Yaskawa INFORM job: OK_R2_O50&56(110_90,0)AWOK.JBI

/JOB
//NAME OK_R2_O50&56(110_90,0)AWOK
///FOLDERNAME X4
//POS
///NPOS 267,267,267,15,0,0
///TOOL 0
///POSTYPE PULSE
///PULSE
C00000=174960,-106597,-120103,3797,95090,-7084
C00001=145956,12891,-49012,9197,114627,-15113
C00002=146175,14682,13914,33266,91894,-54167
C00003=181880,-35169,-29211,31591,75181,-62241
C00004=185949,-21647,605,33162,63920,-63937
C00005=185949,-19989,4400,33558,62671,-64348
C00006=185949,-21647,605,33162,63920,-63937
C00007=186497,-22505,-4,33104,63655,-63786
C00008=185949,-21647,605,33162,63920,-63937
C00009=186993,-19461,2175,32975,63654,-63571
C00010=187282,-18335,3806,33046,63184,-63596
C00011=186993,-19461,2175,32975,63654,-63571
C00012=174899,-22090,-15041,32767,76141,-64809
C00013=150915,-27906,-19346,34122,85374,-71784
C00014=124603,-47737,-34158,-19131,104982,62056
C00015=121442,-51513,-32422,-19687,101389,61480
C00016=118855,-51471,-32397,-20347,100766,60636
C00017=118855,-50574,-30118,-20274,99880,60787
C00018=118855,-51471,-32397,-20347,100766,60636
C00019=121442,-51513,-32422,-19687,101389,61480
C00020=121797,-50324,-29168,-19487,100158,61813
C00021=120620,-50331,-29171,-19792,99877,61431
C00022=121797,-50324,-29168,-19487,100158,61813
C00023=121442,-51513,-32422,-19687,101389,61480
C00024=121603,-51176,-29855,-19536,100099,61752
C00025=121615,-53238,-31000,-19508,99766,61811
C00026=121603,-51176,-29855,-19536,100099,61752
C00027=122128,-47866,-34232,-19785,104374,61232
C00028=84141,-29178,-36607,-14646,114104,67707
C00029=82791,-33286,-36430,-14724,111710,67503
C00030=82229,-34853,-36282,-14765,110740,67415
C00031=82178,-34515,-34630,-14688,109914,67503
C00032=82229,-34853,-36282,-14765,110740,67415
C00033=79147,-30434,-31070,-15425,109262,66446
C00034=78452,-32631,-32544,-15567,108914,66232
C00035=79147,-30434,-31070,-15425,109262,66446
C00036=79730,-28966,-31252,-15378,110209,66539
C00037=81132,-25108,-31519,-15285,112547,66756
C00038=130185,-45166,-65053,-10858,92991,77597
C00039=107206,26705,4589,-9987,92468,27814
C00040=98659,45218,28508,-8039,93095,24888
C00041=98424,43781,30134,-8022,91351,24920
C00042=98486,43736,30153,-8021,91323,24943
C00043=98486,44012,31621,-8015,90571,24990
C00044=98486,43353,27835,-8034,92544,24864
C00045=106492,38043,26451,-21991,88874,27615
C00046=105786,38474,26895,-21964,88638,27404
C00047=106495,38155,26700,-21991,88785,27632
C00048=106495,37420,22299,-22016,90954,27236
C00049=111541,35328,25383,-22123,89542,29330
C00050=102045,-19807,-16561,-21845,84655,26763
C00051=74840,-13391,-38223,-2617,97503,17820
C00052=66507,5010,-12577,6934,97902,16018
C00053=66741,4651,-9261,6890,95673,15973
C00054=66101,6043,-7102,6886,95120,15724
C00055=66101,6129,-6115,6879,94563,15693
C00056=66101,5877,-9999,6916,96808,15817
C00057=80836,-17286,-23478,-14204,80508,20001
C00058=80064,-16344,-22775,-14064,80424,19740
C00059=80850,-17465,-25526,-14169,81645,19874
C00060=68799,5840,-15749,112,106098,15895
C00061=55050,-26211,-40797,-896,104976,11120
C00062=53240,-26394,-33808,-1003,100562,10527
C00063=53174,-26119,-32540,-1008,99922,10509
C00064=53174,-26003,-31510,-1007,99347,10512
C00065=53450,-26813,-34326,-989,100667,10598
C00066=66076,-50527,-45741,-15470,82986,15464
C00067=65365,-49438,-45112,-15396,83017,15209
C00068=66444,-51488,-48366,-15481,84138,15447
C00069=76298,-64666,-67677,-16335,90985,18012
C00070=121005,-146046,-93198,-13283,20086,-50099
C00071=121076,-175637,-121627,-12100,22333,-50657
C00072=121076,-175637,-121627,-12100,22333,-50657
C00073=119842,-145846,-119955,19490,98596,44269
C00074=120072,-86643,-91493,20899,110694,78316
C00075=121200,-92303,-90459,20559,107088,78084
C00076=140479,-121048,-96992,20484,87219,81696
C00077=140479,-120457,-95830,20487,86831,81630
C00078=138616,-107413,-91097,21806,95703,82500
C00079=139134,-110877,-92284,21800,94587,82488
C00080=138616,-107413,-91097,21806,95703,82500
C00081=138504,-107678,-93902,21887,97214,82736
C00082=111033,-68243,-79959,15660,119373,68405
C00083=110238,-79863,-86906,15259,112779,67243
C00084=110238,-79955,-85752,15166,112047,67143
C00085=111039,-68171,-79817,15653,119324,68399
C00086=110811,-71611,-81502,15474,118663,68211
C00087=111039,-68171,-79817,15653,119324,68399
C00088=117681,-73428,-89845,994,113898,68956
C00089=117328,-75555,-88746,937,112132,68814
C00090=117314,-76363,-88422,931,111517,68804
C00091=117314,-76477,-87912,929,111141,68802
C00092=117314,-76038,-89659,939,112445,68812
C00093=117225,-80228,-90181,914,110615,68766
C00094=117357,-73687,-89896,955,113798,68838
C00095=117304,-75426,-92745,956,114658,68828
C00096=117163,-75550,-92733,938,114587,68776
C00097=117163,-75975,-91679,932,113721,68770
C00098=117163,-75740,-92281,935,114212,68773
C00099=117065,-80067,-94252,916,113200,68731
C00100=117163,-75740,-92281,935,114212,68773
C00101=126928,-93462,-104099,-21125,97375,56056
C00102=123436,-95743,-101732,-20630,94052,55403
C00103=119720,-93386,-98939,-20195,92672,54328
C00104=119720,-93542,-97538,-20172,91785,54475
C00105=119720,-93459,-98367,-20185,92306,54389
C00106=117930,-93370,-98332,-19971,91899,53827
C00107=119720,-93459,-98367,-20185,92306,54389
C00108=119671,-100746,-101187,-20141,90406,54690
C00109=119720,-93459,-98367,-20185,92306,54389
C00110=121215,-96042,-102269,-20389,93677,54685
C00111=124737,-93931,-104706,-20902,96960,55358
C00112=120615,-97600,-94225,-24394,68229,41312
C00113=121614,-94302,-98325,-24715,72989,35072
C00114=121413,-94319,-98186,-24655,72844,35027
C00115=121413,-94400,-96939,-24754,72105,35186
C00116=121413,-94319,-98186,-24655,72844,35027
C00117=119573,-94306,-98179,-23998,72315,34443
C00118=121413,-94319,-98186,-24655,72844,35027
C00119=131582,-92162,-101045,-27739,78553,37534
C00120=149979,-79190,-101251,-32758,90741,41130
C00121=131734,108486,68329,-27886,77598,37823
C00122=131746,115175,77213,-28093,75801,38268
C00123=128705,103754,56939,-17355,80936,37498
C00124=126391,103513,58781,-16629,79272,36943
C00125=126391,103204,59430,-16657,78740,37018
C00126=126391,103325,59164,-16645,78953,36987
C00127=131461,101888,64135,-32515,75623,37675
C00128=130460,102804,65331,-32242,75027,37451
C00129=132956,104856,68008,-33106,75465,38321
C00130=123747,88520,39161,-14959,81804,36039
C00131=123722,90598,43933,-15013,79993,36251
C00132=123722,90479,44118,-15020,79823,36272
C00133=123708,91557,46446,-15056,78971,36374
C00134=123735,88704,42579,-15029,79860,36272
C00135=122122,90222,44481,-14459,79203,35813
C00136=121873,91643,46282,-14382,78796,35780
C00137=122407,90627,44476,-14554,79458,35880
C00138=127598,110669,63569,-17480,87727,36370
C00139=127458,127775,88290,-17571,81562,37206
C00140=126717,107110,60862,-17217,87970,36047
C00141=121872,67125,15966,-8400,79107,26604
C00142=119947,67807,18007,-7580,78039,26067
C00143=121767,74654,26232,-6383,76292,25284
C00144=123564,69808,18958,-7132,78404,25740
C00145=121169,67878,17908,-8113,78241,26441
C00146=120006,67962,18206,-7608,78000,26088
C00147=117920,61625,14270,-6708,77001,25483
C00148=118781,60315,11658,-7068,77995,25701
C00149=123961,59152,819,-9198,84481,26863
C00150=132618,-110497,-108947,-28734,74981,37704
C00151=124566,-101520,-102656,-26093,73034,35072
C00152=121381,-96484,-98543,-24994,72121,34061
C00153=122368,-97019,-90544,-25347,66960,42290
C00154=120612,-98338,-92224,-24658,66756,41637
C00155=120867,-94519,-89971,-24653,67354,41604
C00156=120867,-94608,-89971,-24661,67311,41612
C00157=126048,-45476,-69322,-31035,100254,58694
C00158=113068,-21387,-59721,-17378,114816,66130
C00159=116612,-26582,-62582,-17226,114626,67431
C00160=116612,-22676,-66743,-18014,118989,66712
C00161=96791,-67830,-88966,-12124,96584,58954
C00162=98008,-71855,-88035,-12234,94161,59592
C00163=126837,-94677,-94277,-15990,96379,69031
C00164=126113,-98665,-96629,-15951,95659,68871
C00165=124903,-86613,-90535,-14366,101584,74527
C00166=124985,-88200,-92279,-14134,101025,73532
C00167=124953,-89747,-92480,-14095,100368,73599
C00168=120613,-99078,-98492,-7508,100072,69302
C00169=121484,-95136,-96163,-7500,100739,69561
C00170=172923,-99546,-90349,-10002,102117,90375
C00171=179538,-101142,-90555,-8602,100288,90316
C00172=174679,-92302,-94882,-9461,106868,88107
C00173=153430,-78772,-107192,1998,100273,82038
C00174=120149,-70168,-111353,20212,74375,72326
C00175=120057,-133921,-120473,34069,36215,62022
C00176=120146,-106815,-117651,27009,46787,66237
C00177=120793,-117832,-87628,5856,54262,-2374
C00178=128370,-47930,-37102,5352,91873,-78331
C00179=120655,-51136,-30966,4745,86952,-81146
C00180=120656,-51126,-30961,4745,86954,-81145
C00181=121240,-72948,-42427,4950,70443,-81585
C00182=120654,-52833,-32998,4744,87329,-81132
C00183=120662,-49043,-29779,4745,87295,-81131
C00184=130317,-72190,-42085,4090,70120,-78412
C00185=120656,-51164,-30982,4745,86947,-81145
C00186=120655,-51174,-30987,4745,86946,-81146
C00187=120663,-45936,-34749,4755,91934,-80956
C00188=120658,-53922,-38518,-13016,106165,78731
C00189=120658,-51068,-30928,-12795,103038,79070
C00190=123140,-68547,-43521,-11941,93024,80951
C00191=120664,-48985,-29748,-12815,103375,79036
C00192=120728,-51718,-32595,-12818,103725,79022
C00193=121911,-67959,-43086,-12159,93263,80503
C00194=120658,-51052,-30919,-12796,103041,79070
C00195=120658,-51066,-30927,-12796,103039,79070
C00196=93952,-51121,-30967,-10241,104523,-67822
C00197=93953,-51118,-30965,-10240,104524,-67822
C00198=95953,-52479,-31764,-9588,104560,-67115
C00199=94418,-49164,-29853,-10109,104897,-67688
C00200=92862,-50813,-31445,-10614,104829,-68238
C00201=95353,-51547,-30566,-9769,104235,-67302
C00202=95660,-51090,-34260,-9806,106744,-67396
C00203=98759,-53921,-36367,-8775,106946,-66293
C00204=98759,-54646,-38349,-8822,107784,-66355
C00205=121493,-81341,-55216,-13751,94719,44592
C00206=118132,-76574,-45148,-14317,90501,43918
C00207=115160,-74416,-40204,-14849,88108,43182
C00208=114252,-83925,-43808,-15028,85362,43206
C00209=116252,-82247,-47187,-14646,88567,43499
C00210=104568,-69110,-41017,-10991,94760,66686
C00211=117881,-67291,-35412,-18417,97772,58786
C00212=118181,-64547,-30170,-18236,96112,59145
C00213=119086,-67759,-38180,-18148,99432,58962
C00214=99157,-63031,-38155,-9295,97620,77423
C00215=97075,-63253,-34423,-7859,95812,79428
C00216=112438,-76763,-40744,-15729,87696,68197
C00217=115058,-74375,-45131,-15033,92201,68959
C00218=115008,-93546,-53723,-13756,68589,42068
C00219=110722,-90500,-49153,-11979,66777,40535
C00220=111868,-81050,-45580,-11848,69542,40663
C00221=112821,-83961,-50903,-11792,71421,40812
C00222=114232,-64224,-42018,-11630,76204,40845
C00223=113444,-62205,-36873,-11683,74004,40779
C00224=113880,-54019,-32519,-11636,75564,40784
C00225=113879,-55267,-35641,-11577,76817,40664
C00226=113966,-53043,-33005,-11293,67484,41540
C00227=114081,-51287,-29697,-11408,66388,41691
C00228=112504,-67647,-30362,-12654,40215,43900
C00229=111272,-77572,-36344,-12238,37781,43569
C00230=113557,-84331,-43308,-13484,38921,44582
C00231=133973,-53757,-47716,-12346,87026,46675
C00232=129752,5359,-5798,-12169,90869,44838
C00233=101428,28800,15882,-9988,85688,35567
C00234=103132,47107,43189,-16119,89135,35884
C00235=100143,49200,50190,-13622,86051,35125
C00236=98641,51005,54413,-12708,84422,34725
C00237=99366,66814,75390,-15750,91168,34462
C00238=98992,74868,80904,-12799,90779,34103
C00239=96791,41543,38982,-5928,76991,34003
C00240=98035,44299,47107,-8962,72776,34795
C00241=97372,38141,42507,-6482,63971,34987
C00242=99362,40552,35719,-9033,78286,34857
C00243=111144,20698,6526,-10204,87348,38221
C00244=130084,-64485,-54304,2273,113857,-54958
C00245=135702,-112222,-73528,4007,100958,-53286
C00246=120769,-181151,-111215,-14764,18314,-76550
C00247=120640,-138568,-90587,-5858,51266,-81202
C00248=123296,-138495,-91633,-6738,52143,-80161
C00249=127835,-135270,-88085,-8356,52033,-78278
C00250=120633,-141342,-91187,-5942,50214,-81142
C00251=120643,-139926,-92272,-5831,51603,-81221
C00252=119128,-135636,-87879,-5329,51004,-81810
C00253=119353,-140064,-93937,-5303,52463,-81795
C00254=87690,-33642,-44364,-11014,113634,-77986
C00255=119308,-165881,-106719,-1996,57355,-72009
C00256=109869,-45866,-56966,18045,115487,-59616
C00257=82210,-34231,-41337,-6720,113366,-72375
C00258=80442,-31753,-36915,-7087,111776,-72939
C00259=92021,-40775,-43268,-14809,105929,-86070
C00260=92046,-42831,-43945,-14754,105311,-85981
C00261=94159,-47819,-46911,-16507,102203,-90111
C00262=101806,-49911,-44305,-27618,98824,-86333
C00263=105788,-49005,-47861,-27451,102505,-85673
C00264=116531,-78838,-75191,-26148,107297,-82591
C00265=116616,-76076,-73924,-26238,107901,-82700
C00266=-643,-91494,-100294,-9175,50730,69485
BC00000=361150,428180,482576
BC00001=361150,403754,311764
BC00002=327913,423351,363029
BC00003=361483,358049,263035
BC00004=367043,358049,377779
BC00005=367043,358049,377779
BC00006=367043,358049,377779
BC00007=367043,358049,377779
BC00008=367043,358049,377779
BC00009=367043,358049,377779
BC00010=367043,358049,377779
BC00011=367043,358049,377779
BC00012=367043,358049,377779
BC00013=367043,380359,484293
BC00014=282936,371604,325865
BC00015=282936,371604,325865
BC00016=282936,371604,325865
BC00017=282936,371604,325865
BC00018=282936,371604,325865
BC00019=277464,371604,325865
BC00020=280542,371604,325865
BC00021=282936,371604,325865
BC00022=282936,371604,325865
BC00023=282936,371604,325865
BC00024=282936,371604,325865
BC00025=282936,371604,325865
BC00026=282936,371604,325865
BC00027=282936,371604,325865
BC00028=306629,368674,249887
BC00029=306629,368674,249887
BC00030=304240,368674,249887
BC00031=304240,368674,249887
BC00032=304240,368674,249887
BC00033=304240,368674,249887
BC00034=304240,368674,249887
BC00035=304240,368674,249887
BC00036=304240,368674,249887
BC00037=304240,368674,249887
BC00038=315459,352679,342587
BC00039=320619,375147,251105
BC00040=306153,375147,251105
BC00041=306153,375147,251105
BC00042=306153,375147,251105
BC00043=306153,375147,251105
BC00044=306153,375147,251105
BC00045=306153,375147,251105
BC00046=306153,375147,251105
BC00047=306153,375147,251105
BC00048=306153,375147,251105
BC00049=306153,375147,336320
BC00050=266333,375147,400082
BC00051=266333,375147,251105
BC00052=266333,375147,251105
BC00053=266333,375147,251105
BC00054=263944,375147,251105
BC00055=263944,375147,251105
BC00056=263944,375147,251105
BC00057=263944,375147,251105
BC00058=263944,375147,251105
BC00059=263944,375147,251105
BC00060=263944,375147,251105
BC00061=263944,375147,251105
BC00062=263944,375147,251105
BC00063=263944,375147,251105
BC00064=263944,375147,251105
BC00065=263944,375147,251105
BC00066=263944,375147,251105
BC00067=263944,375147,251105
BC00068=263944,375147,251105
BC00069=266333,375147,251105
BC00070=337511,493980,354567
BC00071=337511,493980,1074774
BC00072=337511,493980,1074774
BC00073=22790,343034,1075139
BC00074=22790,343034,1075139
BC00075=22790,343034,1075139
BC00076=22790,343034,1075138
BC00077=22790,343034,1075138
BC00078=22790,343034,1075138
BC00079=22790,343034,1075138
BC00080=22790,343034,1075138
BC00081=22790,343034,1075138
BC00082=22790,343034,1075139
BC00083=22790,343034,1075139
BC00084=22790,343034,1075139
BC00085=22790,343034,1075139
BC00086=22790,343034,1075139
BC00087=22790,343034,1075139
BC00088=22790,343034,1075139
BC00089=22790,343034,1075139
BC00090=22790,343034,1075139
BC00091=22790,343034,1075139
BC00092=22790,343034,1075139
BC00093=22790,343034,1075139
BC00094=22790,343034,1075139
BC00095=60904,322682,1075139
BC00096=60904,322682,1075139
BC00097=60904,322682,1075139
BC00098=60904,322682,1075139
BC00099=60904,322682,1075139
BC00100=60904,322682,1075139
BC00101=33815,332722,1075139
BC00102=33815,332722,1075139
BC00103=33815,332722,1075139
BC00104=33815,332722,1075139
BC00105=33815,332722,1075139
BC00106=33815,332722,1075139
BC00107=33815,332722,1075139
BC00108=33815,332722,1075139
BC00109=33815,332722,1075139
BC00110=33815,332722,1075139
BC00111=33815,332722,1075139
BC00112=24136,376845,1075139
BC00113=29559,333250,1075139
BC00114=29559,333250,1075139
BC00115=29559,333250,1075139
BC00116=29559,333250,1075139
BC00117=29559,333250,1075139
BC00118=29559,333250,1075139
BC00119=29559,333250,1075139
BC00120=29559,333250,1075139
BC00121=29559,516509,1075139
BC00122=47577,452718,1075136
BC00123=47577,442938,1075136
BC00124=47577,442938,1075136
BC00125=47577,442938,1075136
BC00126=47577,442938,1075136
BC00127=47577,442938,1075136
BC00128=47577,442937,1075133
BC00129=47577,442937,1075133
BC00130=47577,442937,1075133
BC00131=47577,442937,1075130
BC00132=47577,442937,1075130
BC00133=47577,442937,1075130
BC00134=47577,442937,1075130
BC00135=47577,442937,1075130
BC00136=47577,442937,1075130
BC00137=47577,442937,1075130
BC00138=47577,442937,1075127
BC00139=47577,442937,1075127
BC00140=47577,430287,1075127
BC00141=47577,430287,1075127
BC00142=47577,430287,1075127
BC00143=47577,430287,1075123
BC00144=47577,430287,1075123
BC00145=47577,430287,1075127
BC00146=47577,430287,1075127
BC00147=47577,430287,1075127
BC00148=47577,430287,1075127
BC00149=47577,430286,1075124
BC00150=30649,324485,1075139
BC00151=30649,324485,1075139
BC00152=30649,324485,1075139
BC00153=31886,372494,1075139
BC00154=31886,372494,1075139
BC00155=31850,371066,1075139
BC00156=31850,371066,1075139
BC00157=31850,371066,1075139
BC00158=31850,371066,1075139
BC00159=31850,371066,1075139
BC00160=33443,371066,1075139
BC00161=1592,351341,1075139
BC00162=1592,351341,1075138
BC00163=1592,353281,1075139
BC00164=1592,353281,1075139
BC00165=1592,351341,1075135
BC00166=774,350737,1075135
BC00167=774,350737,1075135
BC00168=7894,344467,1075139
BC00169=7894,344467,1075139
BC00170=774,350737,1075135
BC00171=774,350737,1075135
BC00172=774,350737,1075135
BC00173=9356,387327,1026996
BC00174=22790,444602,951645
BC00175=22790,500058,951645
BC00176=22790,516485,951645
BC00177=349249,463181,500053
BC00178=347527,372563,432729
BC00179=350010,391797,408474
BC00180=349323,395397,384839
BC00181=349049,396837,375386
BC00182=349049,396837,375386
BC00183=349049,396837,375386
BC00184=349049,396837,375386
BC00185=336040,395438,384865
BC00186=336726,391838,408499
BC00187=336726,391838,408499
BC00188=360192,359857,356751
BC00189=361876,365188,338255
BC00190=362550,367321,330856
BC00191=362550,367321,330856
BC00192=362550,367321,330856
BC00193=366214,367311,331486
BC00194=367653,365171,339250
BC00195=365969,359839,357747
BC00196=354044,349567,361241
BC00197=351834,354289,341394
BC00198=350950,356178,333455
BC00199=350950,356178,333455
BC00200=350950,356178,333455
BC00201=353731,356165,317149
BC00202=354214,355610,318161
BC00203=357589,349550,340448
BC00204=357589,349550,340448
BC00205=357589,349550,340448
BC00206=357589,349550,340448
BC00207=356034,349550,340448
BC00208=355996,349550,340448
BC00209=355996,349550,340448
BC00210=355996,349550,340448
BC00211=355996,349550,340448
BC00212=355996,349550,340448
BC00213=355996,349550,340448
BC00214=355996,349550,340448
BC00215=355996,349550,340448
BC00216=355996,349550,340448
BC00217=355996,349550,340448
BC00218=355996,349550,340447
BC00219=355996,349550,340447
BC00220=355996,349550,340447
BC00221=355996,349550,340447
BC00222=355996,349550,340447
BC00223=355996,349550,340447
BC00224=355996,349550,340447
BC00225=355996,349550,340447
BC00226=355996,349550,340447
BC00227=355996,349550,340447
BC00228=355996,349551,340447
BC00229=355996,349550,340447
BC00230=357589,349550,340447
BC00231=357589,349550,340447
BC00232=357589,349550,340447
BC00233=301964,368322,340447
BC00234=301964,368322,340447
BC00235=301964,368321,340446
BC00236=301964,368321,340446
BC00237=301964,368321,340446
BC00238=301964,368321,340446
BC00239=301964,368321,340446
BC00240=301964,368321,340446
BC00241=301964,368321,340446
BC00242=301964,368321,340446
BC00243=301964,368321,340446
BC00244=354044,349567,455896
BC00245=354044,409351,471270
BC00246=124898,440412,239624
BC00247=124898,382668,239624
BC00248=125863,382654,202128
BC00249=125863,382654,202128
BC00250=125863,382654,202128
BC00251=125863,382654,202128
BC00252=170910,382516,202043
BC00253=155996,382506,212747
BC00254=117092,382506,212747
BC00255=238355,382506,212747
BC00256=238355,382506,212747
BC00257=117092,382506,212747
BC00258=117092,382506,212747
BC00259=117092,382506,212747
BC00260=117092,382506,212747
BC00261=117092,382506,212747
BC00262=117092,382506,212747
BC00263=117092,382506,212747
BC00264=117092,382506,212747
BC00265=117092,489983,212747
BC00266=157445,523407,215162
EC00000=-798156,-183832
EC00001=-798156,-183832
EC00002=-798156,-183832
EC00003=-798156,-183832
EC00004=-798156,-183832
EC00005=-798156,-183832
EC00006=-798156,-183832
EC00007=-798156,-183832
EC00008=-798156,-183832
EC00009=-798156,-183832
EC00010=-798156,-183832
EC00011=-798156,-183832
EC00012=-798156,-183832
EC00013=-798156,-183832
EC00014=-798156,-183832
EC00015=-798156,-183832
EC00016=-798156,-183832
EC00017=-798156,-183832
EC00018=-798156,-183832
EC00019=-798156,-183832
EC00020=-798156,-183832
EC00021=-798156,-183832
EC00022=-798156,-183832
EC00023=-798156,-183832
EC00024=-798156,-183832
EC00025=-798156,-183832
EC00026=-798156,-183832
EC00027=-798156,-183832
EC00028=-798156,-183832
EC00029=-798156,-183832
EC00030=-798156,-183832
EC00031=-798156,-183832
EC00032=-798156,-183832
EC00033=-798156,-183832
EC00034=-798156,-183832
EC00035=-798156,-183832
EC00036=-798156,-183832
EC00037=-798156,-183832
EC00038=-798156,-183832
EC00039=-798156,-183832
EC00040=-798156,-183832
EC00041=-798156,-183832
EC00042=-798156,-183832
EC00043=-798156,-183832
EC00044=-798156,-183832
EC00045=-798156,-183832
EC00046=-798156,-183832
EC00047=-798156,-183832
EC00048=-798156,-183832
EC00049=-798156,-183832
EC00050=-798156,-183832
EC00051=-798156,-183832
EC00052=-798156,-183832
EC00053=-798156,-183832
EC00054=-798156,-183832
EC00055=-798156,-183832
EC00056=-798156,-183832
EC00057=-798156,-183832
EC00058=-798156,-183832
EC00059=-798156,-183832
EC00060=-798156,-183832
EC00061=-798156,-183832
EC00062=-798156,-183832
EC00063=-798156,-183832
EC00064=-798156,-183832
EC00065=-798156,-183832
EC00066=-798156,-183832
EC00067=-798156,-183832
EC00068=-798156,-183832
EC00069=-798156,-183832
EC00070=-798156,-183832
EC00071=-798156,-183832
EC00072=-975524,-183832
EC00073=-975524,-183832
EC00074=-975524,-183832
EC00075=-975524,-183832
EC00076=-975522,-183833
EC00077=-975522,-183833
EC00078=-975522,-183833
EC00079=-975522,-183833
EC00080=-975522,-183833
EC00081=-975522,-183833
EC00082=-975524,-183832
EC00083=-975524,-183832
EC00084=-975524,-183832
EC00085=-975524,-183832
EC00086=-975524,-183832
EC00087=-975524,-183832
EC00088=-975524,-183832
EC00089=-975524,-183832
EC00090=-975524,-183832
EC00091=-975524,-183832
EC00092=-975524,-183832
EC00093=-975524,-183832
EC00094=-975524,-183832
EC00095=-975524,-183832
EC00096=-975524,-183832
EC00097=-975524,-183832
EC00098=-975524,-183832
EC00099=-975524,-183832
EC00100=-975524,-183832
EC00101=-975524,-183832
EC00102=-975524,-183832
EC00103=-975524,-183832
EC00104=-975524,-183832
EC00105=-975524,-183832
EC00106=-975524,-183832
EC00107=-975524,-183832
EC00108=-975524,-183832
EC00109=-975524,-183832
EC00110=-975524,-183832
EC00111=-975524,-183832
EC00112=-975524,-183832
EC00113=-975524,-183832
EC00114=-975524,-183832
EC00115=-975524,-183832
EC00116=-975524,-183832
EC00117=-975524,-183832
EC00118=-975524,-183832
EC00119=-975524,-183832
EC00120=-798157,-183832
EC00121=-798157,-183832
EC00122=-798155,-183833
EC00123=-798155,-183833
EC00124=-798155,-183833
EC00125=-798155,-183833
EC00126=-798155,-183833
EC00127=-798155,-183833
EC00128=-798154,-183833
EC00129=-798154,-183833
EC00130=-798154,-183833
EC00131=-798153,-183833
EC00132=-798153,-183833
EC00133=-798153,-183833
EC00134=-798153,-183833
EC00135=-798153,-183833
EC00136=-798153,-183833
EC00137=-798153,-183833
EC00138=-798152,-183834
EC00139=-798152,-183834
EC00140=-798152,-183834
EC00141=-798152,-183834
EC00142=-798151,-183835
EC00143=-798151,-183834
EC00144=-798151,-183834
EC00145=-798152,-183834
EC00146=-798152,-183834
EC00147=-798152,-183834
EC00148=-798152,-183834
EC00149=-798151,-183834
EC00150=-975524,-183832
EC00151=-975524,-183832
EC00152=-975524,-183832
EC00153=-975524,-183832
EC00154=-975524,-183832
EC00155=-975524,-183832
EC00156=-975524,-183832
EC00157=-975524,-183832
EC00158=-975524,-183832
EC00159=-975524,-183832
EC00160=-975524,-183832
EC00161=-975524,-183832
EC00162=-975522,-183834
EC00163=-975524,-183832
EC00164=-975524,-183832
EC00165=-975521,-183833
EC00166=-975521,-183833
EC00167=-975521,-183833
EC00168=-975524,-183832
EC00169=-975524,-183832
EC00170=-975521,-183833
EC00171=-975521,-183833
EC00172=-975521,-183833
EC00173=-975522,-183833
EC00174=-975524,-183832
EC00175=-975524,-183832
EC00176=-798156,-183832
EC00177=-798156,-183832
EC00178=-798156,-183832
EC00179=-798156,-183832
EC00180=-798156,-183832
EC00181=-798156,-183832
EC00182=-798156,-183832
EC00183=-798156,-183832
EC00184=-798156,-183832
EC00185=-798156,-183832
EC00186=-798156,-183832
EC00187=-798156,-183832
EC00188=-798156,-183832
EC00189=-798156,-183832
EC00190=-798156,-183832
EC00191=-798156,-183832
EC00192=-798156,-183832
EC00193=-798155,-183833
EC00194=-798156,-183832
EC00195=-798156,-183832
EC00196=-798156,-183832
EC00197=-798156,-183832
EC00198=-798156,-183832
EC00199=-798156,-183832
EC00200=-798156,-183832
EC00201=-798156,-183832
EC00202=-798156,-183832
EC00203=-798156,-183832
EC00204=-798156,-183832
EC00205=-798156,-183832
EC00206=-798156,-183832
EC00207=-798156,-183832
EC00208=-798156,-183832
EC00209=-798156,-183832
EC00210=-798156,-183832
EC00211=-798156,-183832
EC00212=-798156,-183832
EC00213=-798156,-183832
EC00214=-798156,-183832
EC00215=-798156,-183832
EC00216=-798156,-183832
EC00217=-798156,-183832
EC00218=-798155,-183832
EC00219=-798155,-183832
EC00220=-798155,-183832
EC00221=-798155,-183832
EC00222=-798155,-183832
EC00223=-798155,-183832
EC00224=-798155,-183832
EC00225=-798155,-183832
EC00226=-798155,-183832
EC00227=-798155,-183832
EC00228=-798152,-183835
EC00229=-798155,-183832
EC00230=-798155,-183832
EC00231=-798155,-183832
EC00232=-798155,-183832
EC00233=-798155,-183832
EC00234=-798155,-183832
EC00235=-798154,-183832
EC00236=-798154,-183832
EC00237=-798154,-183832
EC00238=-798154,-183832
EC00239=-798154,-183832
EC00240=-798154,-183832
EC00241=-798154,-183832
EC00242=-798154,-183832
EC00243=-798154,-183832
EC00244=-798156,-183832
EC00245=-798156,-183832
EC00246=-798156,-183832
EC00247=-798156,-183832
EC00248=-798156,-183832
EC00249=-798156,-183832
EC00250=-798156,-183832
EC00251=-798156,-183832
EC00252=-798156,-183832
EC00253=-798156,-183832
EC00254=-798156,-183832
EC00255=-798156,-183832
EC00256=-798156,-183832
EC00257=-798156,-183832
EC00258=-798156,-183832
EC00259=-798156,-183832
EC00260=-798156,-183832
EC00261=-798156,-183832
EC00262=-798156,-183832
EC00263=-798156,-183832
EC00264=-798156,-183832
EC00265=-798156,-183832
EC00266=-798156,-183832
///POSTYPE BASE
///RECTAN
///RCONF 0,0,0,0,1,0,0,0,0,0,0,0,0,0,0,0,0,0,0,0,0,0,0,0
P00006=2.006,1.622,-0.565,0.0000,0.0000,0.0000
///RCONF 0,0,0,0,0,0,0,0,0,0,0,0,0,0,0,0,0,0,0,0,0,0,0,0
P00023=-2.957,-4.083,2.762,0.0000,0.0000,0.0000
P00024=-1.466,-0.226,-0.419,0.0000,0.0000,0.0000
P00025=3.643,0.007,-2.585,0.0000,0.0000,0.0000
P00031=-0.170,0.039,-0.647,0.0000,0.0000,0.0000
P00032=-0.423,0.157,3.222,0.0000,0.0000,0.0000
P00033=0.854,-1.099,3.047,0.0000,0.0000,0.0000
///RCONF 0,0,0,0,1,0,0,0,0,0,0,0,0,0,0,0,0,0,0,0,0,0,0,0
P00034=-8.151,9.743,-4.393,0.0000,0.0000,0.0000
///RCONF 0,0,0,0,0,0,0,0,0,0,0,0,0,0,0,0,0,0,0,0,0,0,0,0
P00040=2.716,-0.016,3.014,0.0000,0.0000,0.0000
P00044=-8.560,-7.557,-5.232,0.0000,0.0000,0.0000
P00050=-0.123,2.174,-1.314,0.0000,0.0000,0.0000
P00051=-5.945,4.696,-10.293,0.0000,0.0000,0.0000
P00052=-0.153,5.586,-7.982,0.0000,0.0000,0.0000
P00060=1524.284,698.404,-261.973,-0.4635,36.8346,-1.2388
P00061=1211.499,975.999,-261.374,0.5148,35.2356,175.5099
//INST
///DATE 2024/11/25 20:09
///ATTR SC,RW
///GROUP1 RB1,BS1
///GROUP2 ST1
NOP
'OK_r2_O50&56(110_90,0)
'Down
MOVJ C00000 BC00000 VJ=100.00  +MOVJ EC00000 VJ=100.00
MOVJ C00001 BC00001 VJ=100.00  +MOVJ EC00001 VJ=100.00
'Path S1597
SFTOF3D
SFTOF3D
MOVJ C00002 BC00002 VJ=100.00  +MOVJ EC00002 VJ=100.00
MOVL C00003 BC00003 V=333.3  +MOVJ EC00003 VJ=100.00
SMOVL C00004 BC00004 V=100.0  +MOVJ EC00004
SREFP 3 C00005 BC00005  +REFP EC00005
CALL JOB:SEARCH-R1-S13D
SET P025 P006
SFTON3D P025
SMOVL C00006 BC00006 V=100.0  +MOVJ EC00006
SREFP 3 C00007 BC00007  +REFP EC00007
CALL JOB:SEARCH-R1-S13D
SET P025 P006
SFTON3D P025
SMOVL C00008 BC00008 V=100.0  +MOVJ EC00008
SMOVL C00009 BC00009 V=100.0  +MOVJ EC00009
SREFP 3 C00010 BC00010  +REFP EC00010
CALL JOB:SEARCH-R1-S13D
SET P025 P006
SFTON3D P025
SMOVL C00011 BC00011 V=100.0  +MOVJ EC00011
MOVL C00012 BC00012 V=400.0  +MOVJ EC00012 VJ=100.00
MOVL C00013 BC00013 V=1000.0  +MOVJ EC00013 VJ=100.00
'Path S1599
SFTOF3D
MOVJ C00014 BC00014 VJ=100.00  +MOVJ EC00014 VJ=100.00
SMOVL C00015 BC00015 V=333.3  +MOVJ EC00015
SMOVL C00016 BC00016 V=100.0  +MOVJ EC00016
SREFP 3 C00017 BC00017  +REFP EC00017
CALL JOB:SEARCH-R1-S13D
SET P023 P006
SFTON3D P023
SMOVL C00018 BC00018 V=100.0  +MOVJ EC00018
SMOVL C00019 BC00019 V=166.7  +MOVJ EC00019
SMOVL C00020 BC00020 V=100.0  +MOVJ EC00020
SREFP 3 C00021 BC00021  +REFP EC00021
CALL JOB:SEARCH-R1-S13D
SET P023 P006
SFTON3D P023
SMOVL C00022 BC00022 V=100.0  +MOVJ EC00022
SMOVL C00023 BC00023 V=166.7  +MOVJ EC00023
SMOVL C00024 BC00024 V=100.0  +MOVJ EC00024
SREFP 3 C00025 BC00025  +REFP EC00025
CALL JOB:SEARCH-R1-S13D
SET P023 P006
SFTON3D P023
SMOVL C00026 BC00026 V=100.0  +MOVJ EC00026
MOVL C00027 BC00027 V=1000.0  +MOVJ EC00027 VJ=100.00
'Path S1600
SFTOF3D
MOVJ C00028 BC00028 VJ=100.00  +MOVJ EC00028 VJ=100.00
MOVL C00029 BC00029 V=400.0  +MOVJ EC00029 VJ=100.00
SMOVL C00030 BC00030 V=100.0  +MOVJ EC00030
SREFP 3 C00031 BC00031  +REFP EC00031
CALL JOB:SEARCH-R1-S13D
SET P024 P006
SFTON3D P024
SMOVL C00032 BC00032 V=100.0  +MOVJ EC00032
SMOVL C00033 BC00033 V=100.0  +MOVJ EC00033
SREFP 3 C00034 BC00034  +REFP EC00034
CALL JOB:SEARCH-R1-S13D
SET P024 P006
SFTON3D P024
SMOVL C00035 BC00035 V=100.0  +MOVJ EC00035
MOVL C00036 BC00036 V=400.0  +MOVJ EC00036 VJ=100.00
MOVL C00037 BC00037 V=1000.0  +MOVJ EC00037 VJ=100.00
MOVJ C00038 BC00038 VJ=100.00  +MOVJ EC00038 VJ=100.00
'Path S1601
SFTOF3D
MOVJ C00039 BC00039 VJ=100.00  +MOVJ EC00039 VJ=40.00
MOVJ C00040 BC00040 VJ=15.00  +MOVJ EC00040 VJ=40.00
MOVJ C00041 BC00041 VJ=10.00  +MOVJ EC00041 VJ=40.00
SMOVL C00042 BC00042 V=100.0  +MOVJ EC00042
SREFP 3 C00043 BC00043  +REFP EC00043
CALL JOB:SEARCH-R1-S13D
SET P050 P006
SFTON3D P050
SMOVL C00044 BC00044 V=83.3  +MOVJ EC00044
SMOVL C00045 BC00045 V=83.3  +MOVJ EC00045
SREFP 3 C00046 BC00046  +REFP EC00046
CALL JOB:SEARCH-R1-S13D
SET P050 P006
SFTON3D P050
SFTOF3D
SMOVL C00047 BC00047 V=100.0  +MOVJ EC00047
MOVJ C00048 BC00048 VJ=100.00  +MOVJ EC00048 VJ=10.00
MOVJ C00049 BC00049 VJ=100.00  +MOVJ EC00049 VJ=10.00
MOVJ C00050 BC00050 VJ=100.00  +MOVJ EC00050 VJ=50.00
MOVJ C00051 BC00051 VJ=100.00  +MOVJ EC00051 VJ=50.00
MOVJ C00052 BC00052 VJ=100.00  +MOVJ EC00052 VJ=50.00
MOVJ C00053 BC00053 VJ=10.00  +MOVJ EC00053 VJ=50.00
SMOVL C00054 BC00054 V=100.0  +MOVJ EC00054
SREFP 3 C00055 BC00055  +REFP EC00055
CALL JOB:SEARCH-R1-S13D
SET P051 P006
SFTON3D P051
SMOVL C00056 BC00056 V=83.3  +MOVJ EC00056
SMOVL C00057 BC00057 V=100.0  +MOVJ EC00057
SREFP 3 C00058 BC00058  +REFP EC00058
CALL JOB:SEARCH-R1-S13D
SET P051 P006
SFTON3D P051
SFTOF3D
SMOVL C00059 BC00059 V=133.3  +MOVJ EC00059
MOVJ C00060 BC00060 VJ=40.00  +MOVJ EC00060 VJ=40.00
MOVJ C00061 BC00061 VJ=100.00  +MOVJ EC00061 VJ=10.00
MOVJ C00062 BC00062 VJ=10.00  +MOVJ EC00062 VJ=40.00
SMOVL C00063 BC00063 V=100.0  +MOVJ EC00063
SREFP 3 C00064 BC00064  +REFP EC00064
CALL JOB:SEARCH-R1-S13D
SET P052 P006
SFTON3D P052
SMOVL C00065 BC00065 V=83.3  +MOVJ EC00065
SMOVL C00066 BC00066 V=100.0  +MOVJ EC00066
SREFP 3 C00067 BC00067  +REFP EC00067
CALL JOB:SEARCH-R1-S13D
SET P052 P006
SFTON3D P052
SFTOF3D
SMOVL C00068 BC00068 V=100.0  +MOVJ EC00068
MOVJ C00069 BC00069 VJ=100.00  +MOVJ EC00069 VJ=10.00
MOVJ C00070 BC00070 VJ=100.00  +MOVJ EC00070 VJ=100.00
MOVJ C00071 BC00071 VJ=100.00  +MOVJ EC00071 VJ=100.00
MOVJ C00072 BC00072 VJ=100.00  +MOVJ EC00072 VJ=100.00
'Up
MOVJ C00073 BC00073 VJ=100.00  +MOVJ EC00073 VJ=100.00
'Path S1129
SFTOF3D
MOVJ C00074 BC00074 VJ=100.00  +MOVJ EC00074 VJ=100.00
MOVL C00075 BC00075 V=400.0  +MOVJ EC00075 VJ=100.00
SMOVL C00076 BC00076 V=100.0  +MOVJ EC00076
SREFP 3 C00077 BC00077  +REFP EC00077
CALL JOB:SEARCH-R1-S13D
SET P033 P006
SFTON3D P033
SMOVL C00078 BC00078 V=100.0  +MOVJ EC00078
SREFP 3 C00079 BC00079  +REFP EC00079
CALL JOB:SEARCH-R1-S13D
SET P033 P006
SFTON3D P033
SMOVL C00080 BC00080 V=100.0  +MOVJ EC00080
SFTOF3D
SMOVL C00081 BC00081 V=166.7  +MOVJ EC00081
MOVL C00082 BC00082 V=400.0  +MOVJ EC00082 VJ=100.00
SMOVL C00083 BC00083 V=100.0  +MOVJ EC00083
SREFP 3 C00084 BC00084  +REFP EC00084
CALL JOB:SEARCH-R1-S13D
SET P034 P006
SFTON3D P034
SMOVL C00085 BC00085 V=100.0  +MOVJ EC00085
SREFP 3 C00086 BC00086  +REFP EC00086
CALL JOB:SEARCH-R1-S13D
SET P034 P006
SFTON3D P034
SMOVL C00087 BC00087 V=100.0  +MOVJ EC00087
SFTOF3D
MOVJ C00088 BC00088 VJ=100.00  +MOVJ EC00088 VJ=100.00
MOVL C00089 BC00089 V=400.0  +MOVJ EC00089 VJ=100.00
SMOVL C00090 BC00090 V=100.0  +MOVJ EC00090
SREFP 3 C00091 BC00091  +REFP EC00091
CALL JOB:SEARCH-R1-S13D
SET P032 P006
SFTON3D P032
SMOVL C00092 BC00092 V=100.0  +MOVJ EC00092
SREFP 3 C00093 BC00093  +REFP EC00093
CALL JOB:SEARCH-R1-S13D
SET P032 P006
SFTON3D P032
SMOVL C00094 BC00094 V=100.0  +MOVJ EC00094
SFTOF3D
MOVL C00095 BC00095 V=400.0  +MOVJ EC00095 VJ=100.00
SMOVL C00096 BC00096 V=100.0  +MOVJ EC00096
SREFP 3 C00097 BC00097  +REFP EC00097
CALL JOB:SEARCH-R1-S13D
SET P044 P006
SFTON3D P044
SMOVL C00098 BC00098 V=100.0  +MOVJ EC00098
SREFP 3 C00099 BC00099  +REFP EC00099
CALL JOB:SEARCH-R1-S13D
SET P044 P006
SFTON3D P044
SMOVL C00100 BC00100 V=100.0  +MOVJ EC00100
'Path S1118
SFTOF3D
MOVJ C00101 BC00101 VJ=100.00  +MOVJ EC00101 VJ=100.00
MOVL C00102 BC00102 V=400.0  +MOVJ EC00102 VJ=100.00
SMOVL C00103 BC00103 V=100.0  +MOVJ EC00103
SREFP 3 C00104 BC00104  +REFP EC00104
CALL JOB:SEARCH-R1-S13D
SET P031 P006
SFTON3D P031
SMOVL C00105 BC00105 V=100.0  +MOVJ EC00105
SREFP 3 C00106 BC00106  +REFP EC00106
CALL JOB:SEARCH-R1-S13D
SET P031 P006
SFTON3D P031
SMOVL C00107 BC00107 V=100.0  +MOVJ EC00107
SREFP 3 C00108 BC00108  +REFP EC00108
CALL JOB:SEARCH-R1-S13D
SET P031 P006
SFTON3D P031
SMOVL C00109 BC00109 V=100.0  +MOVJ EC00109
MOVL C00110 BC00110 V=400.0  +MOVJ EC00110 VJ=100.00
MOVL C00111 BC00111 V=1000.0  +MOVJ EC00111 VJ=100.00
'Path W344
SFTOF3D
MOVJ C00112 BC00112 VJ=100.00  +MOVJ EC00112 VJ=100.00
SMOVL C00113 BC00113 V=400.0  +MOVJ EC00113
SMOVL C00114 BC00114 V=100.0  +MOVJ EC00114
SREFP 3 C00115 BC00115  +REFP EC00115
CALL JOB:SEARCH-R1-S13D
SET P040 P006
SFTON3D P040
SMOVL C00116 BC00116 V=100.0  +MOVJ EC00116
SREFP 3 C00117 BC00117  +REFP EC00117
CALL JOB:SEARCH-R1-S13D
SET P040 P006
SFTON3D P040
SMOVL C00118 BC00118 V=166.7  +MOVJ EC00118
SFTOF3D
MOVJ C00119 BC00119 VJ=100.00  +MOVJ EC00119 VJ=100.00
MOVJ C00120 BC00120 VJ=100.00  +MOVJ EC00120 VJ=100.00
MOVL C00121 BC00121 V=666.7  +MOVJ EC00121 VJ=100.00
SMOVL C00122 BC00122 V=666.7  +MOVJ EC00122
SMOVL C00123 BC00123 V=400.0  +MOVJ EC00123
SMOVL C00124 BC00124 V=100.0  +MOVJ EC00124
SREFP 3 C00125 BC00125  +REFP EC00125
CALL JOB:SEARCH-R1-S13D
SET P060 P006
SFTON3D P060
SMOVL C00126 BC00126 V=100.0  +MOVJ EC00126
SMOVL C00127 BC00127 V=100.0  +MOVJ EC00127
SREFP 3 C00128 BC00128  +REFP EC00128
CALL JOB:SEARCH-R1-S13D
SET P060 P006
SFTON3D P060
SMOVL C00129 BC00129 V=166.7  +MOVJ EC00129
SFTOF3D
SMOVL C00130 BC00130 V=666.7  +MOVJ EC00130
SMOVL C00131 BC00131 V=400.0  +MOVJ EC00131
SMOVL C00132 BC00132 V=100.0  +MOVJ EC00132
SREFP 3 C00133 BC00133  +REFP EC00133
CALL JOB:SEARCH-R1-S13D
SET P061 P006
SFTON3D P061
SMOVL C00134 BC00134 V=100.0  +MOVJ EC00134
SMOVL C00135 BC00135 V=100.0  +MOVJ EC00135
SREFP 3 C00136 BC00136  +REFP EC00136
CALL JOB:SEARCH-R1-S13D
SET P061 P006
SFTON3D P061
SMOVL C00137 BC00137 V=166.7  +MOVJ EC00137
SFTOF3D
SMOVL C00138 BC00138 V=400.0  +MOVJ EC00138
SMOVL C00139 BC00139 V=400.0  +MOVJ EC00139
SMOVL C00140 BC00140 V=400.0  +MOVJ EC00140
SFTON3D P061
SMOVL C00141 BC00141 V=400.0  +MOVJ EC00141
SMOVL C00142 BC00142 V=166.7 PL=0  +MOVJ EC00142
MACRO1 MJ#(0) ARGF9
ARCON
SMOVL C00143 BC00143 V=10.0  +MOVJ EC00143
ARCOF
SMOVL C00144 BC00144 V=166.7  +MOVJ EC00144
SFTOF3D
SMOVL C00145 BC00145 V=166.7  +MOVJ EC00145
SFTON3D P061
SMOVL C00146 BC00146 V=166.7 PL=0  +MOVJ EC00146
ARCON
SMOVL C00147 BC00147 V=10.0  +MOVJ EC00147
ARCOF
SMOVL C00148 BC00148 V=166.7  +MOVJ EC00148
SFTOF3D
SMOVL C00149 BC00149 V=400.0  +MOVJ EC00149
SMOVL C00150 BC00150 V=1000.0  +MOVJ EC00150
SMOVL C00151 BC00151 V=400.0  +MOVJ EC00151
SMOVL C00152 BC00152 V=166.7 PL=0  +MOVJ EC00152
SREFP 1 C00153 BC00153  +REFP EC00153
SREFP 2 C00154 BC00154  +REFP EC00154
MACRO1 MJ#(0) ARGF9
ARCON
SFTON3D P031
SMOVL C00155 BC00155 V=8.3  +MOVJ EC00155
SMOVC C00156 BC00156 V=8.3  +MOVJ EC00156
SMOVC C00157 BC00157 V=8.3  +MOVJ EC00157
SMOVC C00158 BC00158 V=8.3  +MOVJ EC00158
SMOVL C00159 BC00159 V=8.3  +MOVJ EC00159
ARCOF
SMOVL C00160 BC00160 V=400.0  +MOVJ EC00160
SFTOF3D
SMOVL C00161 BC00161 V=400.0  +MOVJ EC00161
SFTON3D P032
SMOVL C00162 BC00162 V=133.3 PL=0  +MOVJ EC00162
SREFP 1 C00163 BC00163  +REFP EC00163
SREFP 2 C00164 BC00164  +REFP EC00164
MACRO1 MJ#(0) ARGF9
ARCON
SWVON WEV#(60)
SFTON3D P032
SMOVL C00165 BC00165 V=9.2  +MOVJ EC00165
ARCOF
SWVOF
SMOVL C00166 BC00166 V=400.0  +MOVJ EC00166
SFTOF3D
SFTON3D P034
SMOVL C00167 BC00167 V=133.3 PL=0  +MOVJ EC00167
SREFP 1 C00168 BC00168  +REFP EC00168
SREFP 2 C00169 BC00169  +REFP EC00169
MACRO1 MJ#(0) ARGF9
ARCON
SMOVL C00170 BC00170 V=9.2  +MOVJ EC00170
SMOVL C00171 BC00171 V=9.2  +MOVJ EC00171
ARCOF
SMOVL C00172 BC00172 V=400.0  +MOVJ EC00172
SMOVL C00173 BC00173 V=1000.0  +MOVJ EC00173
SFTOF3D
MOVJ C00174 BC00174 VJ=100.00  +MOVJ EC00174 VJ=100.00
MOVJ C00175 BC00175 VJ=100.00  +MOVJ EC00175 VJ=100.00
MOVJ C00176 BC00176 VJ=100.00  +MOVJ EC00176 VJ=100.00
'Down
MOVJ C00177 BC00177 VJ=100.00  +MOVJ EC00177 VJ=100.00
'Path W1603
SFTOF3D
MOVJ C00178 BC00178 VJ=100.00  +MOVJ EC00178 VJ=100.00
'Path W1605
SFTOF3D
SFTON3D P023
MOVJ C00179 BC00179 VJ=100.00  +MOVJ EC00179 VJ=100.00
SMOVL C00180 BC00180 V=1000.0  +MOVJ EC00180
SMOVL C00181 BC00181 V=133.3 PL=0  +MOVJ EC00181
SREFP 1 C00182 BC00182  +REFP EC00182
SREFP 2 C00183 BC00183  +REFP EC00183
MACRO1 MJ#(0) ARGF14
ARCON
SMOVL C00184 BC00184 V=10.8  +MOVJ EC00184
ARCOF
SMOVL C00185 BC00185 V=400.0  +MOVJ EC00185
SMOVL C00186 BC00186 V=1000.0  +MOVJ EC00186
MOVJ C00187 BC00187 VJ=100.00  +MOVJ EC00187 VJ=30.00
SFTOF3D
'Path W1606
SFTOF3D
SFTON3D P024
MOVJ C00188 BC00188 VJ=100.00  +MOVJ EC00188 VJ=100.00
SMOVL C00189 BC00189 V=1000.0  +MOVJ EC00189
SMOVL C00190 BC00190 V=133.3 PL=0  +MOVJ EC00190
SREFP 1 C00191 BC00191  +REFP EC00191
SREFP 2 C00192 BC00192  +REFP EC00192
MACRO1 MJ#(0) ARGF14
ARCON
SMOVL C00193 BC00193 V=11.7  +MOVJ EC00193
ARCOF
SMOVL C00194 BC00194 V=400.0  +MOVJ EC00194
SMOVL C00195 BC00195 V=1000.0  +MOVJ EC00195
SFTOF3D
'Path W1607
SFTOF3D
SFTON3D P024
MOVJ C00196 BC00196 VJ=100.00  +MOVJ EC00196 VJ=100.00
SMOVL C00197 BC00197 V=166.7  +MOVJ EC00197
SMOVL C00198 BC00198 V=133.3 PL=0  +MOVJ EC00198
ARCON
SREFP 1 C00199 BC00199  +REFP EC00199
SREFP 2 C00200 BC00200  +REFP EC00200
MACRO1 MJ#(0) ARGF6
SMOVL C00201 BC00201 V=13.3  +MOVJ EC00201
ARCOF
SMOVL C00202 BC00202 V=400.0  +MOVJ EC00202
SMOVL C00203 BC00203 V=1000.0  +MOVJ EC00203
MOVJ C00204 BC00204 VJ=100.00  +MOVJ EC00204 VJ=30.00
MOVJ C00205 BC00205 VJ=100.00  +MOVJ EC00205 VJ=30.00
MOVJ C00206 BC00206 VJ=30.00  +MOVJ EC00206 VJ=100.00
SFTOF3D
SFTON3D P052
MACRO1 MJ#(0) ARGF14
SMOVL C00207 BC00207 V=83.3  +MOVJ EC00207
ARCON
SMOVL C00208 BC00208 V=10.0  +MOVJ EC00208
ARCOF
SMOVL C00209 BC00209 V=166.7  +MOVJ EC00209
MOVJ C00210 BC00210 VJ=15.00  +MOVJ EC00210 VJ=15.00
MOVL C00211 BC00211 V=133.3  +MOVJ EC00211 VJ=15.00
ARCON
MOVL C00212 BC00212 V=11.7  +MOVJ EC00212 VJ=15.00
ARCOF
MOVL C00213 BC00213 V=166.7  +MOVJ EC00213 VJ=15.00
MOVJ C00214 BC00214 VJ=40.00  +MOVJ EC00214 VJ=70.00
SFTON3D P024
SMOVL C00215 BC00215 V=66.7  +MOVJ EC00215
ARCON
SMOVL C00216 BC00216 V=10.0  +MOVJ EC00216
ARCOF
SMOVL C00217 BC00217 V=250.0  +MOVJ EC00217
SMOVL C00218 BC00218 V=400.0  +MOVJ EC00218
SFTON3D P052
SMOVL C00219 BC00219 V=100.0  +MOVJ EC00219
ARCON
SMOVL C00220 BC00220 V=10.0  +MOVJ EC00220
ARCOF
SMOVL C00221 BC00221 V=166.7  +MOVJ EC00221
SMOVL C00222 BC00222 V=666.7  +MOVJ EC00222
SFTON3D P051
SMOVL C00223 BC00223 V=100.0  +MOVJ EC00223
ARCON
SMOVL C00224 BC00224 V=10.0  +MOVJ EC00224
ARCOF
SMOVL C00225 BC00225 V=333.3  +MOVJ EC00225
SMOVL C00226 BC00226 V=500.0  +MOVJ EC00226
SMOVL C00227 BC00227 V=100.0  +MOVJ EC00227
ARCON
SMOVL C00228 BC00228 V=10.0  +MOVJ EC00228
ARCOF
SMOVL C00229 BC00229 V=166.7  +MOVJ EC00229
SMOVL C00230 BC00230 V=1000.0  +MOVJ EC00230
SMOVL C00231 BC00231 V=1000.0  +MOVJ EC00231
SMOVL C00232 BC00232 V=1000.0  +MOVJ EC00232
SMOVL C00233 BC00233 V=1000.0  +MOVJ EC00233
SMOVL C00234 BC00234 V=400.0  +MOVJ EC00234
SMOVL C00235 BC00235 V=166.7  +MOVJ EC00235
SFTON3D P050
SMOVL C00236 BC00236 V=100.0  +MOVJ EC00236
ARCON
SMOVL C00237 BC00237 V=10.0  +MOVJ EC00237
ARCOF
SMOVL C00238 BC00238 V=133.3  +MOVJ EC00238
SMOVL C00239 BC00239 V=333.3  +MOVJ EC00239
SMOVL C00240 BC00240 V=83.3  +MOVJ EC00240
ARCON
SMOVL C00241 BC00241 V=10.0  +MOVJ EC00241
ARCOF
SMOVL C00242 BC00242 V=83.3  +MOVJ EC00242
MOVJ C00243 BC00243 VJ=100.00  +MOVJ EC00243 VJ=30.00
MOVJ C00244 BC00244 VJ=100.00  +MOVJ EC00244 VJ=100.00
MOVJ C00245 BC00245 VJ=100.00  +MOVJ EC00245 VJ=100.00
MOVJ C00246 BC00246 VJ=100.00  +MOVJ EC00246 VJ=100.00
'Path W1608
SFTOF3D
SFTON3D P025
MOVJ C00247 BC00247 VJ=100.00  +MOVJ EC00247 VJ=100.00
SMOVL C00248 BC00248 V=333.3  +MOVJ EC00248
SMOVL C00249 BC00249 V=133.3 PL=0  +MOVJ EC00249
SREFP 1 C00250 BC00250  +REFP EC00250
SREFP 2 C00251 BC00251  +REFP EC00251
MACRO1 MJ#(0) ARGF14
ARCON
SMOVL C00252 BC00252 V=11.7  +MOVJ EC00252
ARCOF
SMOVL C00253 BC00253 V=400.0  +MOVJ EC00253
SMOVL C00254 BC00254 V=333.3  +MOVJ EC00254
COMM SMOVL C00255 BC00255 V=1000.0  +MOVJ EC00255
COMM SMOVL C00256 BC00256 V=1000.0  +MOVJ EC00256
SMOVL C00257 BC00257 V=166.7  +MOVJ EC00257
ARCON
SMOVL C00258 BC00258 V=12.5  +MOVJ EC00258
ARCOF
SMOVL C00259 BC00259 V=133.3  +MOVJ EC00259
SMOVL C00260 BC00260 V=166.7  +MOVJ EC00260
ARCON
SMOVL C00261 BC00261 V=10.8  +MOVJ EC00261
SMOVL C00262 BC00262 V=10.8  +MOVJ EC00262
ARCOF
SFTOF3D
SMOVL C00263 BC00263 V=250.0  +MOVJ EC00263
SMOVL C00264 BC00264 V=500.0  +MOVJ EC00264
MOVJ C00265 BC00265 VJ=100.00  +MOVJ EC00265 VJ=100.00
MOVJ C00266 BC00266 VJ=100.00  +MOVJ EC00266 VJ=50.00
END
